// TIA Portal V18 export
DATA_BLOCK "UVLamp_DB"   // DB82
VERSION : 0.1
// stored: AutoNumber true, DBAccessibleFromOPCUA true, InstanceOfName UVLamp, InstanceOfType FB
"UVLamp"
   // VAR_INPUT
   //    Emergency : Bool;
   //    MachineStart : Bool;
   //    LampEnable : Bool;
   //    LampMode : Int;
   //    LampSetpointInput : Real;
   //    LampMaintenance : Int;
   //    LampFaultSignal : Bool;
   //    DoorSensor : Bool;
   //    XPosition : DInt;
   //    YPosition : DInt;
   //    WorkingRegionXstart : DInt;
   //    WorkingRegionXend : DInt;
   //    WorkingRegionYstart : DInt;
   //    WorkingRegionYend : DInt;
   //    DevelopmentMode : Bool;
   //    FirstTurnOn : Bool;
   // END_VAR
   // VAR_OUTPUT
   //    LampEnabled : Bool;
   //    LampWorking : Bool;
   //    LampOutONOFF : Bool;
   //    LampDimming : UInt;
   //    LampIntensity : Real;
   //    LampError : Bool;
   //    LampStatus : Int;
   // END_VAR
   // VAR_IN_OUT
   //    LampInONOFF : Bool;
   // END_VAR
   // VAR
   //    InternalWorkingPermission : Bool;
   //    SetpointMax : UInt;
   //    SetpointLimit : UInt;
   //    SetpointConversion : Real;
   //    SetpointOutput : UInt;
   //    SafetyLimitConversion : Real;
   //    IntensityConversion : Real;
   // END_VAR
BEGIN
END_DATA_BLOCK
